(* CODESYS project TicTacToeFredrik.ecp

Project tree, tasks and I/O mapping:
  Controller : 750-8100 PFC100 CS 2ETH ECO, WAGO, order no. 0750-8100, version 5.11.1.16
    application Application
      libraries: 
      task PLC_Task (cyclic, interval t#50ms, priority 15) calls ModBusPOU
      task VISU_TASK (cyclic, interval 100 ms, priority 15) calls nothing
      global variables GVL
      visualisation Visualization
      program TicTacToe_Program [FBD]
      function block TicTacToe [SFC]: Init_entry, End_entry, Init_active, Game_active, Block1_active, Block2_active, Block3_active, Block4_active, Block5_active, Block6_active, Block7_active, Block8_active, Block9_active, Check_active, Check_entry, End_active, BlockInput_active
      program ModBusPOU [ST]
    DeviceAdapter
    Kbus : Kbus, WAGO, version 1.4.0.2
        unmapped channels: K-BUS diagnostics
      Power_Supply_24_VDC : 0750-0602, WAGO, order no. 0750-0602, version 0.0.0.9
        DeviceAdapter
      _8DI_24_VDC_3ms : 0750-0430, WAGO, order no. 0750-0430, version 0.0.0.14
          settings: K-BUS Module slot index = 1
          unmapped channels: _IN
        DeviceAdapter
      _8DO_24_VDC_0_5A : 0750-0530, WAGO, order no. 0750-0530, version 0.0.0.15
          settings: K-BUS Module slot index = 2
          unmapped channels: _OUT
        DeviceAdapter
    MODBUS
      MODBUS : MODBUS, WAGO, order no. n/a, version 1.1.1.15
        _internal_1006_0001_Master : MODBUS Master, WAGO, order no. n/a, version 1.1.1.15
          _internal_1006_0001_IP : MODBUS IP Interface, WAGO, order no. n/a, version 1.1.1.15
              settings: IP settings.Address = '158.38.140.126'
            BECKHOFF_MODBUS_Slave_tcp : MODBUS Remote Slave, WAGO, order no. n/a, version 1.1.1.15
                settings: Slave address / Unit identifier = 1
    Serial
  WAGO_MODBUS_Master : ThirdParty Modbus Master, WAGO, order no. GenericModbusMaster, version 1.0.0.1
    DeviceAdapter
  BECKHOFF_MODBUS_Slave : ThirdParty Modbus Slave, WAGO, order no. GenericModbusSlave, version 1.0.0.0
    DeviceAdapter
  text list GlobalTextList
*)

// Controller/Application/GVL
VAR_GLOBAL
	// Start & Stop
	StartBtn : BOOL;
	StopBtn : BOOL;	
	GameRunning : BOOL;
	GameEnd : BOOL;

	// Buttons
	btn1 : BOOL;
	btn2 : BOOL;
	btn3 : BOOL;
	btn4 : BOOL;
	btn5 : BOOL;
	btn6 : BOOL;
	btn7 : BOOL;
	btn8 : BOOL;
	btn9 : BOOL;
	
	// Text label X
	btn1x : BOOL;
	btn2x : BOOL;
	btn3x : BOOL;
	btn4x : BOOL;
	btn5x : BOOL;
	btn6x : BOOL;
	btn7x : BOOL;
	btn8x : BOOL;
	btn9x : BOOL;
	
	// Text label O
	btn1o : BOOL;
	btn2o : BOOL;
	btn3o : BOOL;
	btn4o : BOOL;
	btn5o : BOOL;
	btn6o : BOOL;
	btn7o : BOOL;
	btn8o : BOOL;
	btn9o : BOOL;
	
	// Won Round
	X_WonRound : BOOL;
	O_WonRound : BOOL;
	Tie : BOOL;
	
	// Whose turn is it?
	TurnX : BOOL;
	TurnO : BOOL;
	
	
	
	
	
	MB5 : BOOL;
	MB6 : BOOL;
	MB7 : BOOL;
	
	// Modbus test variables
	MB1: BOOL;
	MB2: BOOL;
	MB3: BOOL;
	MB4: BOOL;
END_VAR

// Controller/Application/ModBusPOU
PROGRAM ModBusPOU
VAR
END_VAR

MB1;
MB2;
MB3;
MB4;
MB6;
MB7;

END_PROGRAM

// Controller/Application/TicTacToe_Program
PROGRAM TicTacToe_Program
VAR
	TicTacToe: TicTacToe;
END_VAR

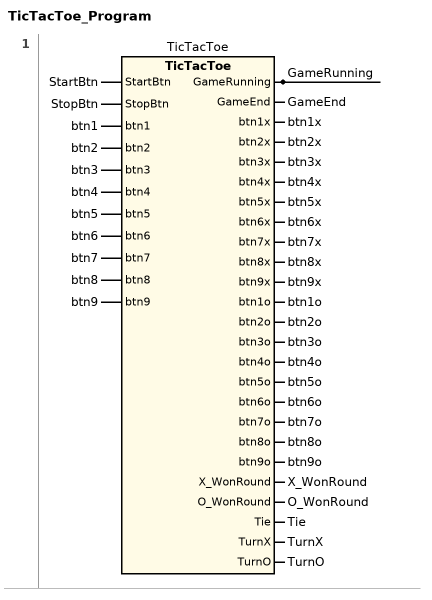
// NETWORK 1
TicTacToe(
    StartBtn := StartBtn,
    StopBtn := StopBtn,
    btn1 := btn1,
    btn2 := btn2,
    btn3 := btn3,
    btn4 := btn4,
    btn5 := btn5,
    btn6 := btn6,
    btn7 := btn7,
    btn8 := btn8,
    btn9 := btn9,
    GameRunning => GameRunning,
    GameEnd => GameEnd,
    btn1x => btn1x,
    btn2x => btn2x,
    btn3x => btn3x,
    btn4x => btn4x,
    btn5x => btn5x,
    btn6x => btn6x,
    btn7x => btn7x,
    btn8x => btn8x,
    btn9x => btn9x,
    btn1o => btn1o,
    btn2o => btn2o,
    btn3o => btn3o,
    btn4o => btn4o,
    btn5o => btn5o,
    btn6o => btn6o,
    btn7o => btn7o,
    btn8o => btn8o,
    btn9o => btn9o,
    X_WonRound => X_WonRound,
    O_WonRound => O_WonRound,
    Tie => Tie,
    TurnX => TurnX,
    TurnO => TurnO);

END_PROGRAM

// Controller/Application/TicTacToe
FUNCTION_BLOCK TicTacToe
VAR_INPUT
	// Start & Stop
	StartBtn : BOOL;
	StopBtn : BOOL;	

	// Buttons
	btn1 : BOOL;
	btn2 : BOOL;
	btn3 : BOOL;
	btn4 : BOOL;
	btn5 : BOOL;
	btn6 : BOOL;
	btn7 : BOOL;
	btn8 : BOOL;
	btn9 : BOOL;
END_VAR
VAR_OUTPUT
	// Game Status
	GameRunning : BOOL;
	GameEnd : BOOL;
	
	// Text label X
	btn1x : BOOL;
	btn2x : BOOL;
	btn3x : BOOL;
	btn4x : BOOL;
	btn5x : BOOL;
	btn6x : BOOL;
	btn7x : BOOL;
	btn8x : BOOL;
	btn9x : BOOL;
	
	// Text label O
	btn1o : BOOL;
	btn2o : BOOL;
	btn3o : BOOL;
	btn4o : BOOL;
	btn5o : BOOL;
	btn6o : BOOL;
	btn7o : BOOL;
	btn8o : BOOL;
	btn9o : BOOL;
	
	// Won Round
	X_WonRound : BOOL;
	O_WonRound : BOOL;
	Tie : BOOL;
	
	//Who's turn is it?
	TurnX : BOOL;
	TurnO : BOOL;
END_VAR
VAR
	// Start & End
	PF_StartGame : BOOL;
	IN_StartGame : BOOL;
	StartGame : BOOL;
	PF_EndGame : BOOL;
	IN_EndGame : BOOL;
	EndGame : BOOL;
	
	// Game
	Turn : INT;
	Progress : BOOL;
	
	// Blocks already used
	Block1_Used : BOOL;
	Block2_Used : BOOL;
	Block3_Used : BOOL;
	Block4_Used : BOOL;
	Block5_Used : BOOL;
	Block6_Used : BOOL;
	Block7_Used : BOOL;
	Block8_Used : BOOL;
	Block9_Used : BOOL;
	
	// Flank detection on the 9 blocks.
	PF_btn1: BOOL;
	IN_btn1: BOOL;
	Signal_btn1: BOOL;
	PF_btn2: BOOL;
	IN_btn2: BOOL;
	Signal_btn2: BOOL;
	PF_btn3: BOOL;
	IN_btn3: BOOL;
	Signal_btn3: BOOL;
	PF_btn4: BOOL;
	IN_btn4: BOOL;
	Signal_btn4: BOOL;
	PF_btn5: BOOL;
	IN_btn5: BOOL;
	Signal_btn5: BOOL;
	PF_btn6: BOOL;
	IN_btn6: BOOL;
	Signal_btn6: BOOL;
	PF_btn7: BOOL;
	IN_btn7: BOOL;
	Signal_btn7: BOOL;
	PF_btn8: BOOL;
	IN_btn8: BOOL;
	Signal_btn8: BOOL;
	PF_btn9: BOOL;
	IN_btn9: BOOL;
	Signal_btn9: BOOL;
END_VAR

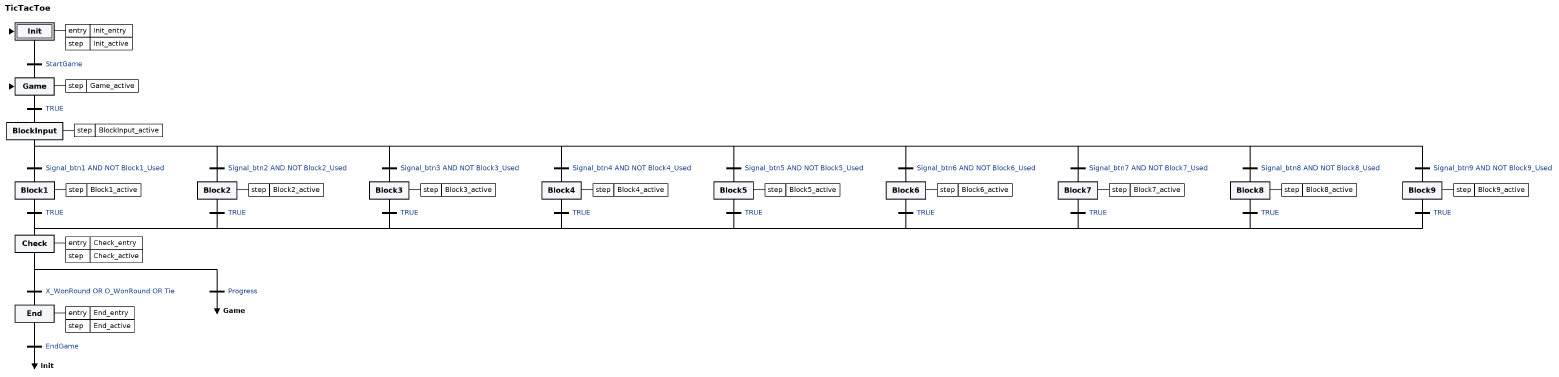
INITIAL_STEP Init:
    Init_entry(P1);  // entry action
    Init_active(N);  // step action
END_STEP
TRANSITION FROM Init TO Game
    := StartGame;
END_TRANSITION
STEP Game:
    Game_active(N);  // step action
END_STEP
TRANSITION FROM Game TO BlockInput
    := TRUE;
END_TRANSITION
STEP BlockInput:
    BlockInput_active(N);  // step action
END_STEP
TRANSITION FROM BlockInput TO Block1
    := Signal_btn1 AND NOT Block1_Used;
END_TRANSITION
STEP Block1:
    Block1_active(N);  // step action
END_STEP
TRANSITION FROM Block1 TO Check
    := TRUE;
END_TRANSITION
TRANSITION FROM BlockInput TO Block2
    := Signal_btn2 AND NOT Block2_Used;
END_TRANSITION
STEP Block2:
    Block2_active(N);  // step action
END_STEP
TRANSITION FROM Block2 TO Check
    := TRUE;
END_TRANSITION
TRANSITION FROM BlockInput TO Block3
    := Signal_btn3 AND NOT Block3_Used;
END_TRANSITION
STEP Block3:
    Block3_active(N);  // step action
END_STEP
TRANSITION FROM Block3 TO Check
    := TRUE;
END_TRANSITION
TRANSITION FROM BlockInput TO Block4
    := Signal_btn4 AND NOT Block4_Used;
END_TRANSITION
STEP Block4:
    Block4_active(N);  // step action
END_STEP
TRANSITION FROM Block4 TO Check
    := TRUE;
END_TRANSITION
TRANSITION FROM BlockInput TO Block5
    := Signal_btn5 AND NOT Block5_Used;
END_TRANSITION
STEP Block5:
    Block5_active(N);  // step action
END_STEP
TRANSITION FROM Block5 TO Check
    := TRUE;
END_TRANSITION
TRANSITION FROM BlockInput TO Block6
    := Signal_btn6 AND NOT Block6_Used;
END_TRANSITION
STEP Block6:
    Block6_active(N);  // step action
END_STEP
TRANSITION FROM Block6 TO Check
    := TRUE;
END_TRANSITION
TRANSITION FROM BlockInput TO Block7
    := Signal_btn7 AND NOT Block7_Used;
END_TRANSITION
STEP Block7:
    Block7_active(N);  // step action
END_STEP
TRANSITION FROM Block7 TO Check
    := TRUE;
END_TRANSITION
TRANSITION FROM BlockInput TO Block8
    := Signal_btn8 AND NOT Block8_Used;
END_TRANSITION
STEP Block8:
    Block8_active(N);  // step action
END_STEP
TRANSITION FROM Block8 TO Check
    := TRUE;
END_TRANSITION
TRANSITION FROM BlockInput TO Block9
    := Signal_btn9 AND NOT Block9_Used;
END_TRANSITION
STEP Block9:
    Block9_active(N);  // step action
END_STEP
TRANSITION FROM Block9 TO Check
    := TRUE;
END_TRANSITION
STEP Check:
    Check_entry(P1);  // entry action
    Check_active(N);  // step action
END_STEP
TRANSITION FROM Check TO End
    := X_WonRound OR O_WonRound OR Tie;
END_TRANSITION
STEP End:
    End_entry(P1);  // entry action
    End_active(N);  // step action
END_STEP
TRANSITION FROM End TO Init
    := EndGame;
END_TRANSITION
TRANSITION FROM Check TO Game
    := Progress;
END_TRANSITION

ACTION Init_entry:
// Sets the StartGame variable to false.
StartGame := FALSE;
END_ACTION

ACTION End_entry:
// Sets the two variables EndGame and GameEnd to FALSE.
EndGame := FALSE;
GameEnd := FALSE;
END_ACTION

ACTION Init_active:
// This is where the game gets initialized, here we among others sets the turn to 1 (since the next turn will be the first one), 
// we resets all variables back to false, this includes the markings and the boolean value of the buttons.
Turn := 1;
X_WonRound := FALSE;
O_WonRound := FALSE;
Tie := FALSE;
EndGame := FALSE;
GameRunning := FALSE;
GameEnd := FALSE;
btn1 := FALSE;
btn2 := FALSE;
btn3 := FALSE;
btn4 := FALSE;
btn5 := FALSE;
btn6 := FALSE;
btn7 := FALSE;
btn8 := FALSE;
btn9 := FALSE;
btn1x := FALSE;
btn2x := FALSE;
btn3x := FALSE;
btn4x := FALSE;
btn5x := FALSE;
btn6x := FALSE;
btn7x := FALSE;
btn8x := FALSE;
btn9x := FALSE;
btn1o := FALSE;
btn2o := FALSE;
btn3o := FALSE;
btn4o := FALSE;
btn5o := FALSE;
btn6o := FALSE;
btn7o := FALSE;
btn8o := FALSE;
btn9o := FALSE;
Signal_btn1 := FALSE;
Signal_btn2 := FALSE;
Signal_btn3 := FALSE;
Signal_btn4 := FALSE;
Signal_btn5 := FALSE;
Signal_btn6 := FALSE;
Signal_btn7 := FALSE;
Signal_btn8 := FALSE;
Signal_btn9 := FALSE;
Block1_Used := FALSE;
Block2_Used := FALSE;
Block3_Used := FALSE;
Block4_Used := FALSE;
Block5_Used := FALSE;
Block6_Used := FALSE;
Block7_Used := FALSE;
Block8_Used := FALSE;
BLock9_Used := FALSE;

// Here we use an positive flank detection on the start button, StartGame is a condition on whether you can move to the next sequence block.
PF_StartGame := StartBtn AND NOT (IN_StartGame);
IN_StartGame := StartBtn;
IF PF_StartGame THEN
	StartGame := TRUE;
END_IF
END_ACTION

ACTION Game_active:
// Sets this variable to true when the game is running.
GameRunning := TRUE;

// Player X have his turn on the turn numbers 1, 3 , 5, 7 and 9
// and the Player O have his turn on the turn numbers 2, 4, 6, 8. 
// This IF-statement checks the turn number and returns who's turn it is.
IF (Turn = 1) OR (Turn = 3) OR (Turn = 5) OR (Turn = 7) OR (Turn = 9) THEN
	TurnX := TRUE;
	TurnO := FALSE;
ELSIF (Turn = 2) OR (Turn = 4) OR (Turn = 6) OR (Turn = 8) THEN
	TurnX := FALSE;
	TurnO := TRUE;
END_IF
END_ACTION

ACTION Block1_active:
// If it's player X's/O's turn, draw an X/O in the block. Tell the game that the block have been used. Then have the turn number increased.
IF TurnX THEN
	btn1x := TRUE;
	// Tegne X i rute 1 => SUNRISE KUKA
	// " NÅ TEGNEST DET " => PI
	
	/// SIGNAL FRA SUNRISE = FERDIG TEGNET => SETT NEXTSTEP TRUE
	
	
	
	ELSIF TurnO THEN
		btn1o := TRUE;
	    // Tegne X i rute 1 => SUNRISE KUKA
	    // " NÅ TEGNEST DET " => PI
	
	    // SIGNAL FRA SUNRISE = FERDIG TEGNET => SETT NEXTSTEP TRUE
END_IF

Block1_Used := TRUE;
Turn := Turn + 1;


//  ----- I BLOKKEN UNDER -----
END_ACTION

ACTION Block2_active:
// If it's player X's/O's turn, draw an X/O in the block. Tell the game that the block have been used. Then have the turn number increased.
IF TurnX THEN
	btn2x := TRUE;
	ELSIF TurnO THEN
		btn2o := TRUE;
END_IF

Block2_Used := TRUE;
Turn := Turn + 1;
END_ACTION

ACTION Block3_active:
// If it's player X's/O's turn, draw an X/O in the block. Tell the game that the block have been used. Then have the turn number increased.
IF TurnX THEN
	btn3x := TRUE;
	ELSIF TurnO THEN
		btn3o := TRUE;
END_IF

Block3_Used := TRUE;
Turn := Turn + 1;
END_ACTION

ACTION Block4_active:
// If it's player X's/O's turn, draw an X/O in the block. Tell the game that the block have been used. Then have the turn number increased.
IF TurnX THEN
	btn4x := TRUE;
	ELSIF TurnO THEN
		btn4o := TRUE;
END_IF

Block4_Used := TRUE;
Turn := Turn + 1;
END_ACTION

ACTION Block5_active:
// If it's player X's/O's turn, draw an X/O in the block. Tell the game that the block have been used. Then have the turn number increased.
IF TurnX THEN
	btn5x := TRUE;
	ELSIF TurnO THEN
		btn5o := TRUE;
END_IF

Block5_Used := TRUE;
Turn := Turn + 1;
END_ACTION

ACTION Block6_active:
// If it's player X's/O's turn, draw an X/O in the block. Tell the game that the block have been used. Then have the turn number increased.
IF TurnX THEN
	btn6x := TRUE;
	ELSIF TurnO THEN
		btn6o := TRUE;
END_IF

Block6_Used := TRUE;
Turn := Turn + 1;
END_ACTION

ACTION Block7_active:
// If it's player X's/O's turn, draw an X/O in the block. Tell the game that the block have been used. Then have the turn number increased.
IF TurnX THEN
	btn7x := TRUE;
	ELSIF TurnO THEN
		btn7o := TRUE;
END_IF

Block7_Used := TRUE;
Turn := Turn + 1;
END_ACTION

ACTION Block8_active:
// If it's player X's/O's turn, draw an X/O in the block. Tell the game that the block have been used. Then have the turn number increased.
IF TurnX THEN
	btn8x := TRUE;
	ELSIF TurnO THEN
		btn8o := TRUE;
END_IF

Block8_Used := TRUE;
Turn := Turn + 1;
END_ACTION

ACTION Block9_active:
// If it's player X's/O's turn, draw an X/O in the block. Tell the game that the block have been used. Then have the turn number increased.
IF TurnX THEN
	btn9x := TRUE;
	ELSIF TurnO THEN
		btn9o := TRUE;
END_IF

Block9_Used := TRUE;
Turn := Turn + 1;
END_ACTION

ACTION Check_active:
(* Here we will check whether not the game is at an end and whether or not anyone have won. 
   We did this by checking every possible outcome of three in a row.
   If X have three in a row, X have won.
   If O have three in a row, O have won.
   If no one have won and the turn number have reached 10 (meaning that 9 turns have been made) then it's a tie. *)

IF (btn1x AND btn2x AND btn3x) OR (btn4x AND btn5x AND btn6x) OR (btn7x AND btn8x AND btn9x) OR (btn1x AND btn5x AND btn9x) OR (btn3x AND btn5x AND btn7x) OR (btn1x AND btn4x AND btn7x) OR (btn2x AND btn5x AND btn8x) OR (btn3x AND btn6x AND btn9x) THEN
	X_WonRound := TRUE;
	O_WonRound := FALSE;
	Tie := FALSE;
	ELSIF (btn1o AND btn2o AND btn3o) OR (btn4o AND btn5o AND btn6o) OR (btn7o AND btn8o AND btn9o) OR (btn1o AND btn5o AND btn9o) OR (btn3o AND btn5o AND btn7o) OR (btn1o AND btn4o AND btn7o) OR (btn2o AND btn5o AND btn8o) OR (btn3o AND btn6o AND btn9o) THEN
	X_WonRound := FALSE;
	O_WonRound := TRUE;
	Tie := FALSE;
	ELSIF Turn = 10 AND NOT X_WonRound AND NOT O_WonRound THEN
	X_WonRound := FALSE;
	O_WonRound := FALSE;
	Tie := TRUE;
	ELSE
		Progress := TRUE;
	END_IF
END_ACTION

ACTION Check_entry:
// Sets the variable Progress to false.
Progress := FALSE;
END_ACTION

ACTION End_active:
// Sets the variable GameEnd to through because the game have come to an end. 
// Flank detection for the Stop button

GameEnd := TRUE;
PF_EndGame := StopBtn AND NOT (IN_EndGame);
IN_EndGame := StopBtn;
IF PF_EndGame THEN
	EndGame := TRUE;
END_IF
END_ACTION

ACTION BlockInput_active:
// Positive flanks for every of the 9 blocks.
PF_btn1 := btn1 AND NOT (IN_btn1);
IN_btn1 := btn1;
Signal_btn1 := PF_btn1;

PF_btn2 := btn2 AND NOT (IN_btn2);
IN_btn2 := btn2;
Signal_btn2 := PF_btn2;

PF_btn3 := btn3 AND NOT (IN_btn3);
IN_btn3 := btn3;
Signal_btn3 := PF_btn3;

PF_btn4 := btn4 AND NOT (IN_btn4);
IN_btn4 := btn4;
Signal_btn4 := PF_btn4;

PF_btn5 := btn5 AND NOT (IN_btn5);
IN_btn5 := btn5;
Signal_btn5 := PF_btn5;

PF_btn6 := btn6 AND NOT (IN_btn6);
IN_btn6 := btn6;
Signal_btn6 := PF_btn6;

PF_btn7 := btn7 AND NOT (IN_btn7);
IN_btn7 := btn7;
Signal_btn7 := PF_btn7;

PF_btn8 := btn8 AND NOT (IN_btn8);
IN_btn8 := btn8;
Signal_btn8 := PF_btn8;

PF_btn9 := btn9 AND NOT (IN_btn9);
IN_btn9 := btn9;
Signal_btn9 := PF_btn9;
END_ACTION

END_FUNCTION_BLOCK

// Controller/Application/Visualization
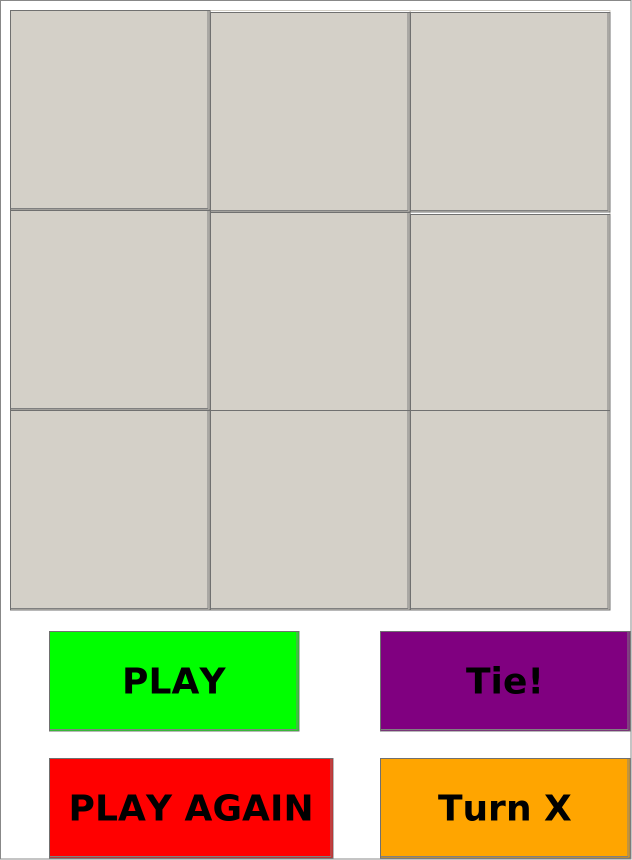
VISUALIZATION Visualization  // 632x860
    Textfield (10,10 200x200), "X", invisible if: NOT GVL.btn1x
    Textfield (210,10 200x200), "X", invisible if: NOT GVL.btn2x
    Textfield (410,10 200x200), "X", invisible if: NOT GVL.btn3x
    Textfield (10,210 200x200), "X", invisible if: NOT GVL.btn4x
    Textfield (210,210 200x200), "X", invisible if: NOT GVL.btn5x
    Textfield (410,210 200x200), "X", invisible if: NOT GVL.btn6x
    Textfield (10,410 200x200), "X", invisible if: NOT GVL.btn7x
    Textfield (210,410 200x200), "X", invisible if: NOT GVL.btn8x
    Textfield (410,410 200x200), "X", invisible if: NOT GVL.btn9x
    Textfield (10,10 200x200), "O", invisible if: NOT GVL.btn1o
    Textfield (210,10 200x200), "O", invisible if: NOT GVL.btn2o
    Textfield (410,14 200x200), "O", invisible if: NOT GVL.btn3o
    Textfield (10,210 200x200), "O", invisible if: NOT GVL.btn4o
    Textfield (210,210 200x200), "O", invisible if: NOT GVL.btn5o
    Textfield (410,210 200x200), "O", invisible if: NOT GVL.btn6o
    Textfield (10,410 200x200), "O", invisible if: NOT GVL.btn7o
    Textfield (210,410 200x200), "O", invisible if: NOT GVL.btn8o
    Textfield (410,410 200x200), "O", invisible if: NOT GVL.btn9o
    Button (10,10 200x200), invisible if: GVL.btn1o or GVL.btn1x
        tap GVL.btn1
    Button (10,210 200x200), invisible if: GVL.btn4o or GVL.btn4x
        tap GVL.btn4
    Button (10,410 200x200), invisible if: GVL.btn7o or GVL.btn7x
        tap GVL.btn7
    Button (210,12 200x200), invisible if: GVL.btn2o or GVL.btn2x
        tap GVL.btn2
    Button (210,212 200x200), invisible if: GVL.btn5o or GVL.btn5x
        tap GVL.btn5
    Button (210,410 200x200), invisible if: GVL.btn8o or GVL.btn8x
        tap GVL.btn8
    Button (410,12 200x200), invisible if: GVL.btn3o or GVL.btn3x
        tap GVL.btn3
    Button (410,214 200x200), invisible if: GVL.btn6o or GVL.btn6x
        tap GVL.btn6
    Button (410,410 200x200), invisible if: GVL.btn9o or GVL.btn9x
        tap GVL.btn9
    Button (49,631 250x100), "PLAY", invisible if: GVL.GameRunning
        tap GVL.StartBtn
    Button (49,758 284x100), "PLAY AGAIN", invisible if: NOT GVL.GameEnd
        tap GVL.StopBtn
    Button (380,631 250x100), "X Won!", invisible if: NOT GVL.X_WonRound
    Button (380,631 250x100), "O Won!", invisible if: NOT GVL.O_WonRound
    Button (380,758 250x100), "Turn O", invisible if: GVL.TurnX OR GVL.O_WonRound OR GVL.X_WonRound OR GVL.Tie OR NOT GVL.GameRunning
    Button (380,758 250x100), "Turn X", invisible if: GVL.TurnO OR GVL.O_WonRound OR GVL.X_WonRound OR GVL.Tie OR NOT GVL.GameRunning
    Button (380,631 250x100), "Tie!", invisible if: NOT GVL.Tie
END_VISUALIZATION
